// TIA Portal V17 export
// export: Created 2026-04-13T11:12:04.6703146Z, ExportSetting WithDefaults, DisplayName Totally Integrated Automation Portal, DisplayVersion V17 Update 4, DisplayName TIA Portal Openness, DisplayVersion V17 Update 4, DisplayName TIA Portal Version Control Interface, DisplayVersion V17, DisplayName SINAMICS Startdrive Advanced, DisplayVersion V17, DisplayName SINAMICS Startdrive G130, G150, S120, S150, SINAMICS MV, S210, DisplayVersion V17, DisplayName SINAMICS Startdrive G110M, G120, G120C, G120D, G120P, G115D, DisplayVersion V17, DisplayName STEP 7 Professional, DisplayVersion V17 Update 4, DisplayName STEP 7 Safety, DisplayVersion V17, DisplayName WinCC Professional, DisplayVersion V17 Update 4
FUNCTION_BLOCK "D3-布袋记录"   // FB74, SCL
{ S7_Optimized_Access := 'TRUE' }
VERSION : 0.1
// stored: AutoNumber true, IsIECCheckEnabled false, IsRetainMemResEnabled false, MemoryReserve 100, SetENOAutomatically false, UDAEnableTagReadback false
   VAR_INPUT
      事件触发器 : Bool;
      清除日志 : Bool;
   END_VAR
   VAR_IN_OUT
      事件记录 : Array[1..20] of String[20];
      事件编号 : Array[1..20] of Int;
      当前记录次数 : Int;
   END_VAR
   VAR
      R_TRIG_Instance { S7_SetPoint := 'True'} : R_TRIG;
      tm_DTL { ExternalAccessible := 'False'; ExternalVisible := 'False'; ExternalWritable := 'False'} : DTL;
   END_VAR
   VAR_TEMP
      tm_Ret : Int;
      tm_i : Int;
      tm_str : String[20];
      tm_year : String[5];
      tm_month : String[3];
      tm_day : String[3];
      tm_hour : String[3];
      tm_minute : String[3];
      tm_second : String[3];
      tm_strcount : String[5];
      tm_strC : String[4];
      tm_empty : Array[1..20] of String[20];
      tm_cempty : Array[1..20] of Int;
   END_VAR
BEGIN
   #R_TRIG_Instance(CLK:=#事件触发器);
   IF #当前记录次数 < 1 THEN
       #当前记录次数 := 1;
   END_IF;

   IF (#当前记录次数 > 9999) OR  #清除日志 THEN
       #当前记录次数 := 1;

       #事件记录 := #tm_empty;
       #事件编号 := #tm_cempty;
       #当前记录次数 := 1;
   END_IF;

   IF #R_TRIG_Instance.Q THEN
       #tm_Ret := RD_LOC_T(#tm_DTL);
       #tm_year := UINT_TO_STRING(#tm_DTL.YEAR);
       #tm_month := USINT_TO_STRING(#tm_DTL.MONTH);
       #tm_day := USINT_TO_STRING(#tm_DTL.DAY);
       #tm_hour := USINT_TO_STRING(#tm_DTL.HOUR+7);
       #tm_minute := USINT_TO_STRING(#tm_DTL.MINUTE);
       #tm_second := USINT_TO_STRING(#tm_DTL.SECOND);
       #tm_str := '';
       #tm_str[1] := #tm_year[2];
       #tm_str[2] := #tm_year[3];
       #tm_str[3] := #tm_year[4];
       #tm_str[4] := #tm_year[5];
       #tm_str[5] := '-';
       IF LEN(#tm_month) = 3 THEN
           #tm_str[6] := #tm_month[2];
           #tm_str[7] := #tm_month[3];
       ELSE
           #tm_str[6] := '0';
           #tm_str[7] := #tm_month[2];
       END_IF;
       #tm_str[8] := '-';
       IF LEN(#tm_day)= 3 THEN
       #tm_str[9] := #tm_day[2];
       #tm_str[10] := #tm_day[3];
   ELSE
       #tm_str[9] := '0';
       #tm_str[10] := #tm_day[2];;
   END_IF;

   #tm_str[11] := ' ';
   IF LEN(#tm_hour) = 3 THEN
       #tm_str[12] := #tm_hour[2];
       #tm_str[13] := #tm_hour[3];
   ELSE
       #tm_str[12] := '0';
       #tm_str[13] := #tm_hour[2];
   END_IF;
   #tm_str[14] := ':';
   IF LEN(#tm_minute) = 3 THEN
       #tm_str[15] := #tm_minute[2];
       #tm_str[16] := #tm_minute[3];
   ELSE
       #tm_str[15] := '0';
       #tm_str[16] := #tm_minute[2];
   END_IF;
       #tm_str[17] := ':';
       IF LEN(#tm_second) = 3 THEN
           #tm_str[18] := #tm_second[2];
           #tm_str[19] := #tm_second[3];
       ELSE
           #tm_str[18] := '0';
           #tm_str[19] := #tm_second[2];
       END_IF;
       #tm_strcount := INT_TO_STRING(#当前记录次数);
       IF LEN(#tm_strcount) = 2 THEN
           #tm_strC[1] := '0';
           #tm_strC[2] := '0';
           #tm_strC[3] := '0';
           #tm_strC[4] := #tm_strcount[2];
       END_IF;

       IF LEN(#tm_strcount) = 3 THEN
           #tm_strC[1] := '0';
           #tm_strC[2] := '0';
           #tm_strC[3] := #tm_strcount[2];
           #tm_strC[4] := #tm_strcount[3];
       END_IF;
       IF LEN(#tm_strcount) = 4 THEN
           #tm_strC[1] := '0';
           #tm_strC[2] := #tm_strcount[2];
           #tm_strC[3] := #tm_strcount[3];
           #tm_strC[4] := #tm_strcount[4];
       END_IF;
       IF LEN(#tm_strcount) =5 THEN
           #tm_strC[1] := #tm_strcount[2];
           #tm_strC[2] := #tm_strcount[3];
           #tm_strC[3] := #tm_strcount[4];
           #tm_strC[4] := #tm_strcount[5];
       END_IF;



       IF #当前记录次数 < 20 THEN
           #事件记录[#当前记录次数] := #tm_str;
           #事件编号[#当前记录次数] :=#当前记录次数;
       ELSE
           FOR #tm_i := 1 TO 19 DO
               #事件编号[#tm_i] := #事件编号[#tm_i + 1];
               #事件编号[#tm_i] := #事件编号[#tm_i + 1];
           END_FOR;
           #事件记录[20] := #tm_str;
           #事件编号[20] := #当前记录次数;
       END_IF;
       #当前记录次数 := #当前记录次数 + 1;
   END_IF;
END_FUNCTION_BLOCK
